// Mitsubishi GX Works2 project: 2023-06-08 #1 생산자동화기능사 13번   PLC: Q03UDV
// 생산자동화기능사

// global labels: Global1
VAR_GLOBAL
  PB1 AT X0 : BOOL;
  PB2 AT X1 : BOOL;
  정지 AT X2 : BOOL;
  공급후진 AT X3 : BOOL;
  공급전진 AT X4 : BOOL;
  가공후진 AT X5 : BOOL;
  가공전진 AT X6 : BOOL;
  송출후진 AT X7 : BOOL;
  송출전진 AT X8 : BOOL;
  배출후진 AT X9 : BOOL;
  배출전진 AT X0A : BOOL;
  매거진 AT X0B : BOOL;
  금속센서 AT X0F : BOOL;
  PB3 AT X0C : BOOL;
  적 AT Y20 : BOOL;
  황 AT Y21 : BOOL;
  녹 AT Y22 : BOOL;
  공급1 AT Y23 : BOOL;
  공급2 AT Y24 : BOOL;
  가공 AT Y25 : BOOL;
  드릴 AT Y26 : BOOL;
  송출 AT Y27 : BOOL;
  배출 AT Y28 : BOOL;
  컨베이어 AT Y29 : BOOL;
END_VAR

PROGRAM 테스트동작
VAR
  PHASE : INT;
END_VAR
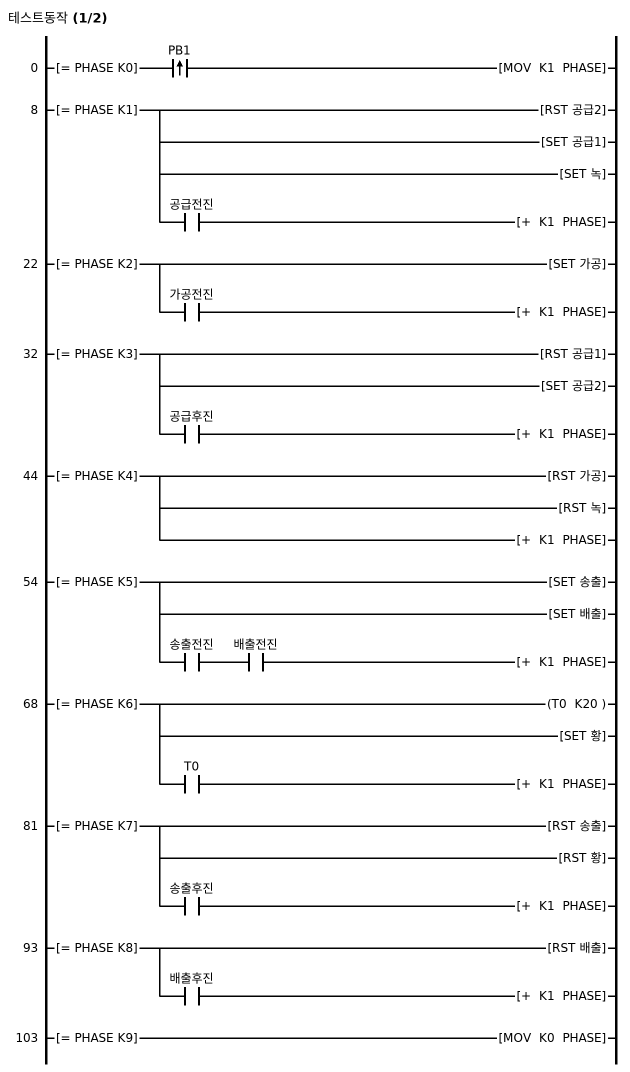
0     LD=     PHASE K0
      ANDP    PB1
      MOV     K1 PHASE
8     LD=     PHASE K1
      RST     공급2
      SET     공급1
      SET     녹
      AND     공급전진
      +       K1 PHASE
22    LD=     PHASE K2
      SET     가공
      AND     가공전진
      +       K1 PHASE
32    LD=     PHASE K3
      RST     공급1
      SET     공급2
      AND     공급후진
      +       K1 PHASE
44    LD=     PHASE K4
      RST     가공
      RST     녹
      +       K1 PHASE
54    LD=     PHASE K5
      SET     송출
      SET     배출
      AND     송출전진
      AND     배출전진
      +       K1 PHASE
68    LD=     PHASE K6
      OUT     T0 K20
      SET     황
      AND     T0
      +       K1 PHASE
81    LD=     PHASE K7
      RST     송출
      RST     황
      AND     송출후진
      +       K1 PHASE
93    LD=     PHASE K8
      RST     배출
      AND     배출후진
      +       K1 PHASE
103   LD=     PHASE K9
      MOV     K0 PHASE
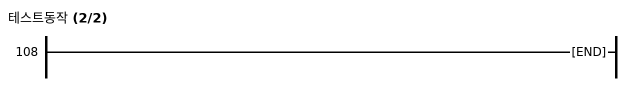
108   END
END_PROGRAM

PROGRAM 생산자동화기능사
VAR
  PHASE : INT;
  MODE : INT;
END_VAR
VAR CONSTANT
  단속 : INT;
  연속 : INT := 1;
END_VAR
VAR
  LOOP : ARRAY [0..0] OF INT;
  METAL : INT;
END_VAR
VAR CONSTANT
  금속 : INT := 1;
  비금속 : INT := 2;
END_VAR
VAR
  BLINK1 : ARRAY [0..3] OF BOOL;
  EMG : INT;
  BLINK2 : ARRAY [0..3] OF BOOL;
END_VAR
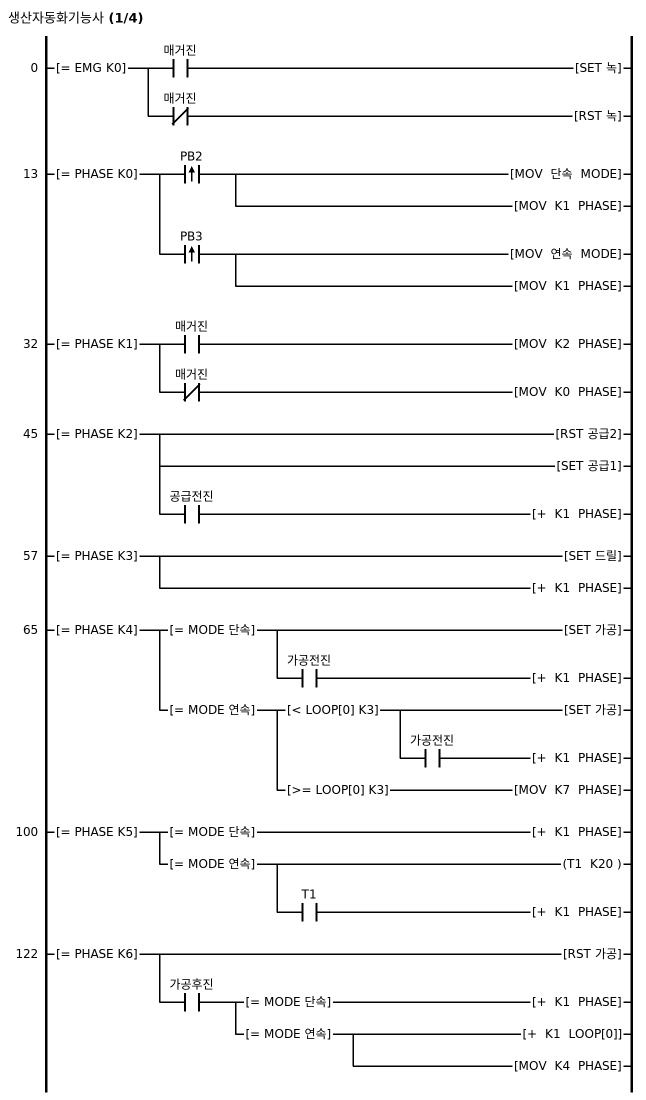
0     LD=     EMG K0
      MPS
      AND     매거진
      SET     녹
      MPP
      ANI     매거진
      RST     녹
13    LD=     PHASE K0
      MPS
      ANDP    PB2
      MOV     단속 MODE
      MOV     K1 PHASE
      MPP
      ANDP    PB3
      MOV     연속 MODE
      MOV     K1 PHASE
32    LD=     PHASE K1
      MPS
      AND     매거진
      MOV     K2 PHASE
      MPP
      ANI     매거진
      MOV     K0 PHASE
45    LD=     PHASE K2
      RST     공급2
      SET     공급1
      AND     공급전진
      +       K1 PHASE
57    LD=     PHASE K3
      SET     드릴
      +       K1 PHASE
65    LD=     PHASE K4
      MPS
      AND=    MODE 단속
      SET     가공
      AND     가공전진
      +       K1 PHASE
      MPP
      AND=    MODE 연속
      MPS
      AND<    LOOP[0] K3
      SET     가공
      AND     가공전진
      +       K1 PHASE
      MPP
      AND>=   LOOP[0] K3
      MOV     K7 PHASE
100   LD=     PHASE K5
      MPS
      AND=    MODE 단속
      +       K1 PHASE
      MPP
      AND=    MODE 연속
      OUT     T1 K20
      AND     T1
      +       K1 PHASE
122   LD=     PHASE K6
      RST     가공
      AND     가공후진
      MPS
      AND=    MODE 단속
      +       K1 PHASE
      MPP
      AND=    MODE 연속
      +       K1 LOOP[0]
      MOV     K4 PHASE
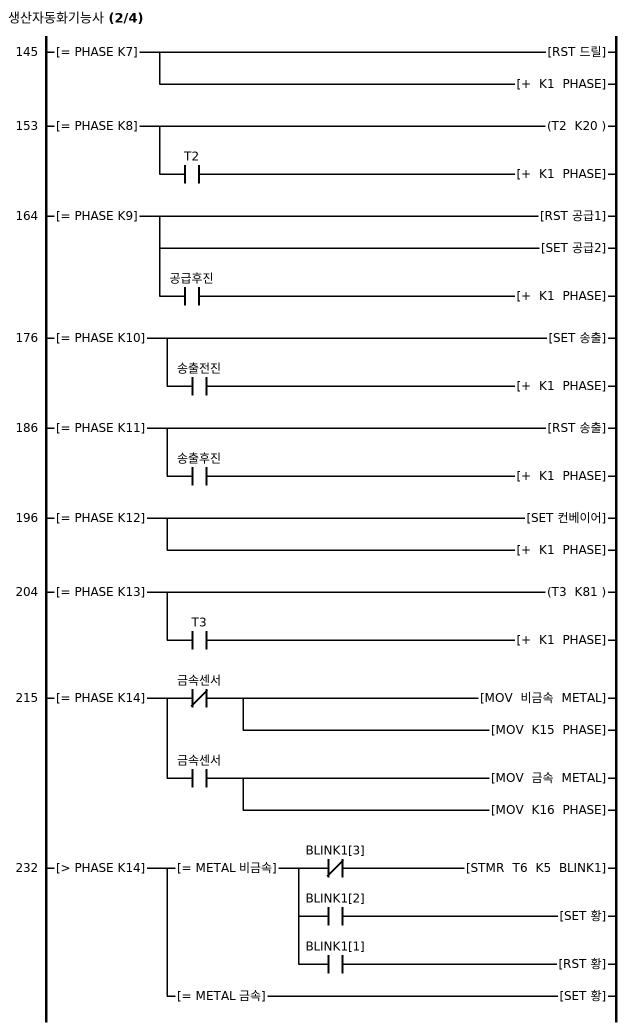
145   LD=     PHASE K7
      RST     드릴
      +       K1 PHASE
153   LD=     PHASE K8
      OUT     T2 K20
      AND     T2
      +       K1 PHASE
164   LD=     PHASE K9
      RST     공급1
      SET     공급2
      AND     공급후진
      +       K1 PHASE
176   LD=     PHASE K10
      SET     송출
      AND     송출전진
      +       K1 PHASE
186   LD=     PHASE K11
      RST     송출
      AND     송출후진
      +       K1 PHASE
196   LD=     PHASE K12
      SET     컨베이어
      +       K1 PHASE
204   LD=     PHASE K13
      OUT     T3 K81
      AND     T3
      +       K1 PHASE
215   LD=     PHASE K14
      MPS
      ANI     금속센서
      MOV     비금속 METAL
      MOV     K15 PHASE
      MPP
      AND     금속센서
      MOV     금속 METAL
      MOV     K16 PHASE
232   LD>     PHASE K14
      MPS
      AND=    METAL 비금속
      MPS
      ANI     BLINK1[3]
      STMR    T6 K5 BLINK1
      MRD
      AND     BLINK1[2]
      SET     황
      MPP
      AND     BLINK1[1]
      RST     황
      MPP
      AND=    METAL 금속
      SET     황
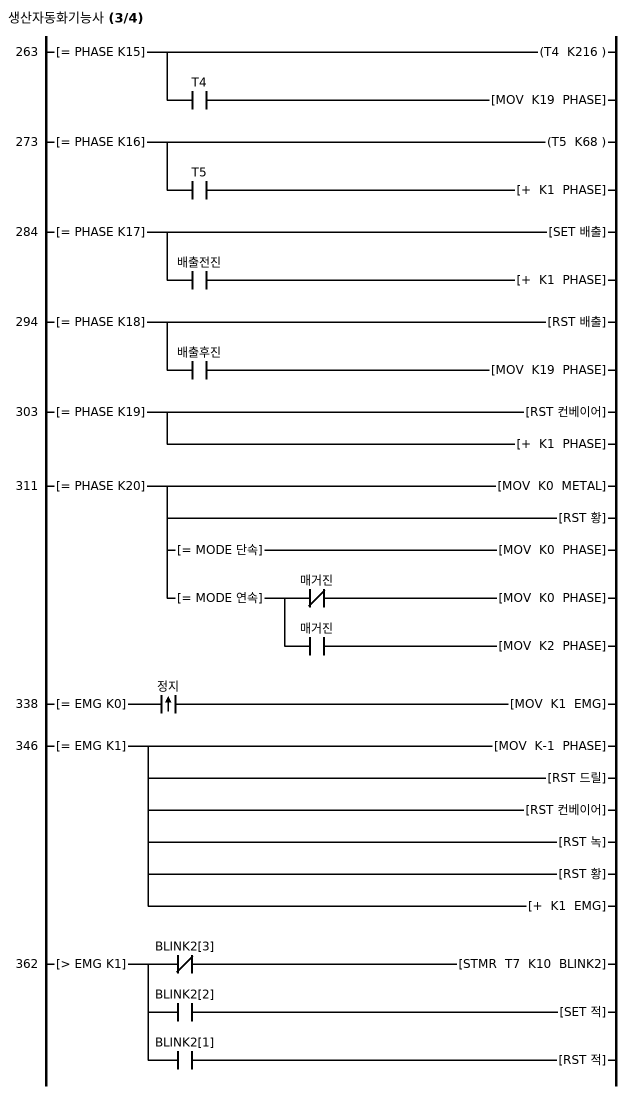
263   LD=     PHASE K15
      OUT     T4 K216
      AND     T4
      MOV     K19 PHASE
273   LD=     PHASE K16
      OUT     T5 K68
      AND     T5
      +       K1 PHASE
284   LD=     PHASE K17
      SET     배출
      AND     배출전진
      +       K1 PHASE
294   LD=     PHASE K18
      RST     배출
      AND     배출후진
      MOV     K19 PHASE
303   LD=     PHASE K19
      RST     컨베이어
      +       K1 PHASE
311   LD=     PHASE K20
      MOV     K0 METAL
      RST     황
      MPS
      AND=    MODE 단속
      MOV     K0 PHASE
      MPP
      AND=    MODE 연속
      MPS
      ANI     매거진
      MOV     K0 PHASE
      MPP
      AND     매거진
      MOV     K2 PHASE
338   LD=     EMG K0
      ANDP    정지
      MOV     K1 EMG
346   LD=     EMG K1
      MOV     K-1 PHASE
      RST     드릴
      RST     컨베이어
      RST     녹
      RST     황
      +       K1 EMG
362   LD>     EMG K1
      MPS
      ANI     BLINK2[3]
      STMR    T7 K10 BLINK2
      MRD
      AND     BLINK2[2]
      SET     적
      MPP
      AND     BLINK2[1]
      RST     적
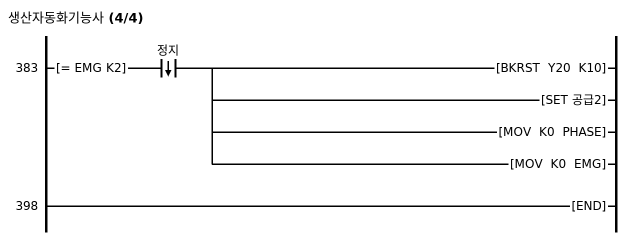
383   LD=     EMG K2
      ANDF    정지
      BKRST   Y20 K10
      SET     공급2
      MOV     K0 PHASE
      MOV     K0 EMG
398   END
END_PROGRAM
